// TwinCAT 3 PLC project PLC_1
// ProgramVersion: 3.1.4024.0
// libraries:
//   Tc2_Standard, * (Beckhoff Automation GmbH)
//   Tc2_System, * (Beckhoff Automation GmbH)
//   Tc2_XmlDataSrv, * (Beckhoff Automation GmbH)
//   Tc3_JsonXml, * (Beckhoff Automation GmbH)
//   Tc3_Module, * (Beckhoff Automation GmbH)
// project tree:
//   DUTs/GenericHierarchyList/GenericHierarchy/ItemCS/Content/DefaultIdentity/ St_DefaultIdentity.TcDUT
//   DUTs/GenericHierarchyList/GenericHierarchy/ItemCS/Content/ItemList/ItemOUT1/Content/DefaultIdentity/ ST_DefaultIdentityOUT1.TcDUT
//   DUTs/GenericHierarchyList/GenericHierarchy/ItemCS/Content/ItemList/ItemOUT1/Content/ItemList/ItemPK1/Identity/ ST_Identity_PK1_OUT1.TcDUT
//   DUTs/GenericHierarchyList/GenericHierarchy/ItemCS/Content/ItemList/ItemOUT1/Content/ItemList/ItemPK1/logs/ ST_logs_PK1_OUT1.TcDUT (not stored)
//   DUTs/GenericHierarchyList/GenericHierarchy/ItemCS/Content/ItemList/ItemOUT1/Content/ItemList/ItemPK1/RejectReason/ ST_RejectReason_PK1_OUT1.TcDUT
//   DUTs/GenericHierarchyList/GenericHierarchy/ItemCS/Content/ItemList/ItemOUT1/Content/ItemList/ItemPK1/ ST_ItemPK1_OUT1.TcDUT
//   DUTs/GenericHierarchyList/GenericHierarchy/ItemCS/Content/ItemList/ItemOUT1/Content/ItemList/ItemPK2/Identity/ ST_Identity_PK2_OUT1.TcDUT
//   DUTs/GenericHierarchyList/GenericHierarchy/ItemCS/Content/ItemList/ItemOUT1/Content/ItemList/ItemPK2/logs/ ST_logs_PK2_OUT1.TcDUT (not stored)
//   DUTs/GenericHierarchyList/GenericHierarchy/ItemCS/Content/ItemList/ItemOUT1/Content/ItemList/ItemPK2/RejectReason/ ST_RejectReason_PK2_OUT1.TcDUT
//   DUTs/GenericHierarchyList/GenericHierarchy/ItemCS/Content/ItemList/ItemOUT1/Content/ItemList/ItemPK2/ ST_ItemPK2_OUT1.TcDUT
//   DUTs/GenericHierarchyList/GenericHierarchy/ItemCS/Content/ItemList/ItemOUT1/Content/ItemList/ItemPK3/Identity/ ST_Identity_PK3_OUT1.TcDUT
//   DUTs/GenericHierarchyList/GenericHierarchy/ItemCS/Content/ItemList/ItemOUT1/Content/ItemList/ItemPK3/logs/ ST_logs_PK3_OUT1.TcDUT (not stored)
//   DUTs/GenericHierarchyList/GenericHierarchy/ItemCS/Content/ItemList/ItemOUT1/Content/ItemList/ItemPK3/RejectReason/ ST_RejectReason_PK3_OUT1.TcDUT
//   DUTs/GenericHierarchyList/GenericHierarchy/ItemCS/Content/ItemList/ItemOUT1/Content/ItemList/ItemPK3/ ST_ItemPK3_OUT1.TcDUT
//   DUTs/GenericHierarchyList/GenericHierarchy/ItemCS/Content/ItemList/ItemOUT1/Content/ItemList/ItemPK4/Identity/ ST_Identity_PK4_OUT1.TcDUT
//   DUTs/GenericHierarchyList/GenericHierarchy/ItemCS/Content/ItemList/ItemOUT1/Content/ItemList/ItemPK4/logs/ ST_logs_PK4_OUT1.TcDUT (not stored)
//   DUTs/GenericHierarchyList/GenericHierarchy/ItemCS/Content/ItemList/ItemOUT1/Content/ItemList/ItemPK4/RejectReason/ ST_RejectReason_PK4_OUT1.TcDUT
//   DUTs/GenericHierarchyList/GenericHierarchy/ItemCS/Content/ItemList/ItemOUT1/Content/ItemList/ItemPK4/ ST_ItemPK4_OUT1.TcDUT
//   DUTs/GenericHierarchyList/GenericHierarchy/ItemCS/Content/ItemList/ItemOUT1/Content/ItemList/ ST_ItemListOUT1.TcDUT
//   DUTs/GenericHierarchyList/GenericHierarchy/ItemCS/Content/ItemList/ItemOUT1/Content/ ST_ContentOUT1.TcDUT
//   DUTs/GenericHierarchyList/GenericHierarchy/ItemCS/Content/ItemList/ItemOUT1/Identity/ ST_IdentityOUT1.TcDUT
//   DUTs/GenericHierarchyList/GenericHierarchy/ItemCS/Content/ItemList/ItemOUT1/logs/ ST_logsOUT1.TcDUT (not stored)
//   DUTs/GenericHierarchyList/GenericHierarchy/ItemCS/Content/ItemList/ItemOUT1/RejectReason/ ST_RejectReasonOUT1.TcDUT
//   DUTs/GenericHierarchyList/GenericHierarchy/ItemCS/Content/ItemList/ItemOUT1/ ST_ItemOUT1.TcDUT
//   DUTs/GenericHierarchyList/GenericHierarchy/ItemCS/Content/ItemList/ItemOUT2/Content/DefaultIdentity/ ST_DefaultIdentityOUT2.TcDUT
//   DUTs/GenericHierarchyList/GenericHierarchy/ItemCS/Content/ItemList/ItemOUT2/Content/ItemList/ItemPK1/Identity/ ST_Identity_PK1_OUT2.TcDUT
//   DUTs/GenericHierarchyList/GenericHierarchy/ItemCS/Content/ItemList/ItemOUT2/Content/ItemList/ItemPK1/logs/ ST_logs_PK1_OUT2.TcDUT (not stored)
//   DUTs/GenericHierarchyList/GenericHierarchy/ItemCS/Content/ItemList/ItemOUT2/Content/ItemList/ItemPK1/RejectReason/ ST_RejectReason_PK1_OUT2.TcDUT
//   DUTs/GenericHierarchyList/GenericHierarchy/ItemCS/Content/ItemList/ItemOUT2/Content/ItemList/ItemPK1/ ST_ItemPK1_OUT2.TcDUT
//   DUTs/GenericHierarchyList/GenericHierarchy/ItemCS/Content/ItemList/ItemOUT2/Content/ItemList/ItemPK2/Identity/ ST_Identity_PK2_OUT2.TcDUT
//   DUTs/GenericHierarchyList/GenericHierarchy/ItemCS/Content/ItemList/ItemOUT2/Content/ItemList/ItemPK2/logs/ ST_logs_PK2_OUT2.TcDUT (not stored)
//   DUTs/GenericHierarchyList/GenericHierarchy/ItemCS/Content/ItemList/ItemOUT2/Content/ItemList/ItemPK2/RejectReason/ ST_RejectReason_PK2_OUT2.TcDUT
//   DUTs/GenericHierarchyList/GenericHierarchy/ItemCS/Content/ItemList/ItemOUT2/Content/ItemList/ItemPK2/ ST_ItemPK2_OUT2.TcDUT
//   DUTs/GenericHierarchyList/GenericHierarchy/ItemCS/Content/ItemList/ItemOUT2/Content/ItemList/ItemPK3/Identity/ ST_Identity_PK3_OUT2.TcDUT
//   DUTs/GenericHierarchyList/GenericHierarchy/ItemCS/Content/ItemList/ItemOUT2/Content/ItemList/ItemPK3/logs/ ST_logs_PK3_OUT2.TcDUT (not stored)
//   DUTs/GenericHierarchyList/GenericHierarchy/ItemCS/Content/ItemList/ItemOUT2/Content/ItemList/ItemPK3/RejectReason/ ST_RejectReason_PK3_OUT2.TcDUT
//   DUTs/GenericHierarchyList/GenericHierarchy/ItemCS/Content/ItemList/ItemOUT2/Content/ItemList/ItemPK3/ ST_ItemPK3_OUT2.TcDUT
//   DUTs/GenericHierarchyList/GenericHierarchy/ItemCS/Content/ItemList/ItemOUT2/Content/ItemList/ItemPK4/Identity/ ST_Identity_PK4_OUT2.TcDUT
//   DUTs/GenericHierarchyList/GenericHierarchy/ItemCS/Content/ItemList/ItemOUT2/Content/ItemList/ItemPK4/logs/ ST_logs_PK4_OUT2.TcDUT (not stored)
//   DUTs/GenericHierarchyList/GenericHierarchy/ItemCS/Content/ItemList/ItemOUT2/Content/ItemList/ItemPK4/RejectReason/ ST_RejectReason_PK4_OUT2.TcDUT
//   DUTs/GenericHierarchyList/GenericHierarchy/ItemCS/Content/ItemList/ItemOUT2/Content/ItemList/ItemPK4/ ST_ItemPK4_OUT2.TcDUT
//   DUTs/GenericHierarchyList/GenericHierarchy/ItemCS/Content/ItemList/ItemOUT2/Content/ItemList/ ST_ItemListOUT2.TcDUT
//   DUTs/GenericHierarchyList/GenericHierarchy/ItemCS/Content/ItemList/ItemOUT2/Content/ ST_ContentOUT2.TcDUT
//   DUTs/GenericHierarchyList/GenericHierarchy/ItemCS/Content/ItemList/ItemOUT2/Identity/ ST_IdentityOUT2.TcDUT
//   DUTs/GenericHierarchyList/GenericHierarchy/ItemCS/Content/ItemList/ItemOUT2/logs/ ST_logsOUT2.TcDUT (not stored)
//   DUTs/GenericHierarchyList/GenericHierarchy/ItemCS/Content/ItemList/ItemOUT2/RejectReason/ ST_RejectReasonOUT2.TcDUT
//   DUTs/GenericHierarchyList/GenericHierarchy/ItemCS/Content/ItemList/ItemOUT2/ ST_ItemOUT2.TcDUT
//   DUTs/GenericHierarchyList/GenericHierarchy/ItemCS/Content/ItemList/ItemOUT3/Content/DefaultIdentity/ ST_DefaultIdentityOUT3.TcDUT
//   DUTs/GenericHierarchyList/GenericHierarchy/ItemCS/Content/ItemList/ItemOUT3/Content/ItemList/ItemPK1/Identity/ ST_Identity_PK1_OUT3.TcDUT
//   DUTs/GenericHierarchyList/GenericHierarchy/ItemCS/Content/ItemList/ItemOUT3/Content/ItemList/ItemPK1/logs/ ST_logs_PK1_OUT3.TcDUT (not stored)
//   DUTs/GenericHierarchyList/GenericHierarchy/ItemCS/Content/ItemList/ItemOUT3/Content/ItemList/ItemPK1/RejectReason/ ST_RejectReason_PK1_OUT3.TcDUT
//   DUTs/GenericHierarchyList/GenericHierarchy/ItemCS/Content/ItemList/ItemOUT3/Content/ItemList/ItemPK1/ ST_ItemPK1_OUT3.TcDUT
//   DUTs/GenericHierarchyList/GenericHierarchy/ItemCS/Content/ItemList/ItemOUT3/Content/ItemList/ItemPK2/Identity/ ST_Identity_PK2_OUT3.TcDUT
//   DUTs/GenericHierarchyList/GenericHierarchy/ItemCS/Content/ItemList/ItemOUT3/Content/ItemList/ItemPK2/logs/ ST_logs_PK2_OUT3.TcDUT (not stored)
//   DUTs/GenericHierarchyList/GenericHierarchy/ItemCS/Content/ItemList/ItemOUT3/Content/ItemList/ItemPK2/RejectReason/ ST_RejectReason_PK2_OUT3.TcDUT
//   DUTs/GenericHierarchyList/GenericHierarchy/ItemCS/Content/ItemList/ItemOUT3/Content/ItemList/ItemPK2/ ST_ItemPK2_OUT3.TcDUT
//   DUTs/GenericHierarchyList/GenericHierarchy/ItemCS/Content/ItemList/ItemOUT3/Content/ItemList/ItemPK3/Identity/ ST_Identity_PK3_OUT3.TcDUT
//   DUTs/GenericHierarchyList/GenericHierarchy/ItemCS/Content/ItemList/ItemOUT3/Content/ItemList/ItemPK3/logs/ ST_logs_PK3_OUT3.TcDUT (not stored)
//   DUTs/GenericHierarchyList/GenericHierarchy/ItemCS/Content/ItemList/ItemOUT3/Content/ItemList/ItemPK3/RejectReason/ ST_RejectReason_PK3_OUT3.TcDUT
//   DUTs/GenericHierarchyList/GenericHierarchy/ItemCS/Content/ItemList/ItemOUT3/Content/ItemList/ItemPK3/ ST_ItemPK3_OUT3.TcDUT
//   DUTs/GenericHierarchyList/GenericHierarchy/ItemCS/Content/ItemList/ItemOUT3/Content/ItemList/ItemPK4/Identity/ ST_Identity_PK4_OUT3.TcDUT
//   DUTs/GenericHierarchyList/GenericHierarchy/ItemCS/Content/ItemList/ItemOUT3/Content/ItemList/ItemPK4/logs/ ST_logs_PK4_OUT3.TcDUT (not stored)
//   DUTs/GenericHierarchyList/GenericHierarchy/ItemCS/Content/ItemList/ItemOUT3/Content/ItemList/ItemPK4/RejectReason/ ST_RejectReason_PK4_OUT3.TcDUT
//   DUTs/GenericHierarchyList/GenericHierarchy/ItemCS/Content/ItemList/ItemOUT3/Content/ItemList/ItemPK4/ ST_ItemPK4_OUT3.TcDUT
//   DUTs/GenericHierarchyList/GenericHierarchy/ItemCS/Content/ItemList/ItemOUT3/Content/ItemList/ ST_ItemListOUT3.TcDUT
//   DUTs/GenericHierarchyList/GenericHierarchy/ItemCS/Content/ItemList/ItemOUT3/Content/ ST_ContentOUT3.TcDUT
//   DUTs/GenericHierarchyList/GenericHierarchy/ItemCS/Content/ItemList/ItemOUT3/Identity/ ST_IdentityOUT3.TcDUT
//   DUTs/GenericHierarchyList/GenericHierarchy/ItemCS/Content/ItemList/ItemOUT3/logs/ ST_logsOUT3.TcDUT (not stored)
//   DUTs/GenericHierarchyList/GenericHierarchy/ItemCS/Content/ItemList/ItemOUT3/RejectReason/ ST_RejectReasonOUT3.TcDUT
//   DUTs/GenericHierarchyList/GenericHierarchy/ItemCS/Content/ItemList/ItemOUT3/ ST_ItemOUT3.TcDUT
//   DUTs/GenericHierarchyList/GenericHierarchy/ItemCS/Content/ItemList/ ST_ItemList.TcDUT
//   DUTs/GenericHierarchyList/GenericHierarchy/ItemCS/Content/ ST_Content.TcDUT
//   DUTs/GenericHierarchyList/GenericHierarchy/ItemCS/Identity/ ST_Identity.TcDUT
//   DUTs/GenericHierarchyList/GenericHierarchy/ItemCS/logs/ ST_logs.TcDUT (not stored)
//   DUTs/GenericHierarchyList/GenericHierarchy/ItemCS/RejectReason/ ST_RejectReason.TcDUT
//   DUTs/GenericHierarchyList/GenericHierarchy/ItemCS/ ST_ItemCS.TcDUT
//   DUTs/GenericHierarchyList/GenericHierarchy/ ST_GenericHierarchy_Write.TcDUT
//   DUTs/GenericHierarchyList/Messageheader/ ST_MessageHeader_Write.TcDUT
//   DUTs/GenericHierarchyList/ ST_GenericHierarchyList.TcDUT
//   DUTs/ProductionChange/PRODUCTINFORMATION/PRODUCT/HIERARCHYDATALIST/HIERARCHYDATACS/ ST_HIERARCHYDATACS.TcDUT
//   DUTs/ProductionChange/PRODUCTINFORMATION/PRODUCT/HIERARCHYDATALIST/HIERARCHYDATAOUT/ ST_HIERARCHYDATAOUT.TcDUT
//   DUTs/ProductionChange/PRODUCTINFORMATION/PRODUCT/HIERARCHYDATALIST/HIERARCHYDATAPK/ ST_HIERARCHYDATAPK.TcDUT
//   DUTs/ProductionChange/PRODUCTINFORMATION/PRODUCT/HIERARCHYDATALIST/ ST_HIERARCHYDATALIST.TcDUT
//   DUTs/ProductionChange/PRODUCTINFORMATION/PRODUCT/ ST_PRODUCT.TcDUT
//   DUTs/ProductionChange/PRODUCTINFORMATION/SETTINGS/TOLERANCETHRESHOLDOUT/ ST_TOLERANCETHRESHOLDOUT.TcDUT
//   DUTs/ProductionChange/PRODUCTINFORMATION/SETTINGS/ ST_SETTINGS.TcDUT
//   DUTs/ProductionChange/PRODUCTINFORMATION/SETTINGS/TOLERANCETHRESHOLDPK/ ST_TOLERANCETHRESHOLDPK.TcDUT
//   DUTs/ProductionChange/PRODUCTINFORMATION/ ST_PRODUCTINFORMATION.TcDUT
//   DUTs/ProductionChange/ ST_MESSAGEHEADER.TcDUT, ST_ProductionChange.TcDUT
//   / PlcTask.TcTTO
//   POUs/ FB_XMLRead.TcPOU, FB_XmlWrite.TcPOU, MAIN.TcPOU
// real-time tasks:
//   TASK PlcTask: cycle T#10ms, priority 20, ADS port 350

CONFIGURATION PLC_1
    RESOURCE PLC ON TwinCAT3
        TASK PlcTask(INTERVAL := T#10ms, PRIORITY := 20);
        PROGRAM MAIN WITH PlcTask : MAIN;
    END_RESOURCE
END_CONFIGURATION

// ---- DUTs/GenericHierarchyList/GenericHierarchy/ItemCS/Content/DefaultIdentity/St_DefaultIdentity.TcDUT
TYPE St_DefaultIdentity :
STRUCT
	SKU					:STRING;
	GTIN				:STRING;
	ProductionOrder		:STRING;
	LocalProductionOrder:STRING;
	PITCode				:STRING;
	BatchID				:STRING;
	ProductionLine		:STRING;
END_STRUCT
END_TYPE

// ---- DUTs/GenericHierarchyList/GenericHierarchy/ItemCS/Content/ItemList/ItemOUT1/Content/DefaultIdentity/ST_DefaultIdentityOUT1.TcDUT
TYPE ST_DefaultIdentityOUT1 :
STRUCT
	SKU						:STRING;
	GTIN					:STRING;
	ProductionOrder			:STRING;
	LocalProductionOrder	:STRING;
	PITCode					:STRING;
	BatchID					:STRING;
	ProductionLine			:STRING;
END_STRUCT
END_TYPE

// ---- DUTs/GenericHierarchyList/GenericHierarchy/ItemCS/Content/ItemList/ItemOUT1/Content/ItemList/ItemPK1/Identity/ST_Identity_PK1_OUT1.TcDUT
TYPE ST_Identity_PK1_OUT1 :
STRUCT
	ID	:STRING;
	ReadQuality:STRING;
END_STRUCT
END_TYPE

// ---- DUTs/GenericHierarchyList/GenericHierarchy/ItemCS/Content/ItemList/ItemOUT1/Content/ItemList/ItemPK1/RejectReason/ST_RejectReason_PK1_OUT1.TcDUT
TYPE ST_RejectReason_PK1_OUT1 :
STRUCT
	Reason	:STRING;
END_STRUCT
END_TYPE

// ---- DUTs/GenericHierarchyList/GenericHierarchy/ItemCS/Content/ItemList/ItemOUT1/Content/ItemList/ItemPK1/ST_ItemPK1_OUT1.TcDUT
TYPE ST_ItemPK1_OUT1 :
STRUCT
	Identity		:ST_Identity_PK1_OUT1;
	ItemState		:STRING;
	RejectReason	:ST_RejectReason_PK1_OUT1;
	logs			:ST_logs_PK1_OUT1;
	NoRead			:STRING;
END_STRUCT
END_TYPE

// ---- DUTs/GenericHierarchyList/GenericHierarchy/ItemCS/Content/ItemList/ItemOUT1/Content/ItemList/ItemPK2/Identity/ST_Identity_PK2_OUT1.TcDUT
TYPE ST_Identity_PK2_OUT1 :
STRUCT
	ID	:STRING;
	ReadQuality:STRING;
END_STRUCT
END_TYPE

// ---- DUTs/GenericHierarchyList/GenericHierarchy/ItemCS/Content/ItemList/ItemOUT1/Content/ItemList/ItemPK2/RejectReason/ST_RejectReason_PK2_OUT1.TcDUT
TYPE ST_RejectReason_PK2_OUT1 :
STRUCT
	Reason	:STRING;
END_STRUCT
END_TYPE

// ---- DUTs/GenericHierarchyList/GenericHierarchy/ItemCS/Content/ItemList/ItemOUT1/Content/ItemList/ItemPK2/ST_ItemPK2_OUT1.TcDUT
TYPE ST_ItemPK2_OUT1 :
STRUCT
	Identity		:ST_Identity_PK2_OUT1;
	ItemState		:STRING;
	RejectReason	:ST_RejectReason_PK2_OUT1;
	logs			:ST_logs_PK2_OUT1;
	NoRead			:STRING;
END_STRUCT
END_TYPE

// ---- DUTs/GenericHierarchyList/GenericHierarchy/ItemCS/Content/ItemList/ItemOUT1/Content/ItemList/ItemPK3/Identity/ST_Identity_PK3_OUT1.TcDUT
TYPE ST_Identity_PK3_OUT1 :
STRUCT
	ID	:STRING;
	ReadQuality:STRING;
END_STRUCT
END_TYPE

// ---- DUTs/GenericHierarchyList/GenericHierarchy/ItemCS/Content/ItemList/ItemOUT1/Content/ItemList/ItemPK3/RejectReason/ST_RejectReason_PK3_OUT1.TcDUT
TYPE ST_RejectReason_PK3_OUT1 :
STRUCT
	Reason	:STRING;
END_STRUCT
END_TYPE

// ---- DUTs/GenericHierarchyList/GenericHierarchy/ItemCS/Content/ItemList/ItemOUT1/Content/ItemList/ItemPK3/ST_ItemPK3_OUT1.TcDUT
TYPE ST_ItemPK3_OUT1 :
STRUCT
	Identity		:ST_Identity_PK3_OUT1;
	ItemState		:STRING;
	RejectReason	:ST_RejectReason_PK3_OUT1;
	logs			:ST_logs_PK3_OUT1;
	NoRead			:STRING;
END_STRUCT
END_TYPE

// ---- DUTs/GenericHierarchyList/GenericHierarchy/ItemCS/Content/ItemList/ItemOUT1/Content/ItemList/ItemPK4/Identity/ST_Identity_PK4_OUT1.TcDUT
TYPE ST_Identity_PK4_OUT1 :
STRUCT
	ID	:STRING;
	ReadQuality:STRING;
END_STRUCT
END_TYPE

// ---- DUTs/GenericHierarchyList/GenericHierarchy/ItemCS/Content/ItemList/ItemOUT1/Content/ItemList/ItemPK4/RejectReason/ST_RejectReason_PK4_OUT1.TcDUT
TYPE ST_RejectReason_PK4_OUT1 :
STRUCT
	Reason	:STRING;
END_STRUCT
END_TYPE

// ---- DUTs/GenericHierarchyList/GenericHierarchy/ItemCS/Content/ItemList/ItemOUT1/Content/ItemList/ItemPK4/ST_ItemPK4_OUT1.TcDUT
TYPE ST_ItemPK4_OUT1 :
STRUCT
	Identity		:ST_Identity_PK4_OUT1;
	ItemState		:STRING;
	RejectReason	:ST_RejectReason_PK4_OUT1;
	logs			:ST_logs_PK4_OUT1;
	NoRead			:STRING;
END_STRUCT
END_TYPE

// ---- DUTs/GenericHierarchyList/GenericHierarchy/ItemCS/Content/ItemList/ItemOUT1/Content/ItemList/ST_ItemListOUT1.TcDUT
TYPE ST_ItemListOUT1 :
STRUCT
	ItemPK1 	:ST_ItemPK1_OUT1;
	ItemPK2 	:ST_ItemPK2_OUT1;
	ItemPK3 	:ST_ItemPK3_OUT1;
	ItemPK4 	:ST_ItemPK4_OUT1;
END_STRUCT
END_TYPE

// ---- DUTs/GenericHierarchyList/GenericHierarchy/ItemCS/Content/ItemList/ItemOUT1/Content/ST_ContentOUT1.TcDUT
TYPE ST_ContentOUT1 :
STRUCT
	DefaultIdentity   :ST_DefaultIdentityOUT1;
	ExpectedItemCount	:STRING;
	ItemReadRate		:STRING;
	ItemList			:ST_ItemListOUT1;
END_STRUCT
END_TYPE

// ---- DUTs/GenericHierarchyList/GenericHierarchy/ItemCS/Content/ItemList/ItemOUT1/Identity/ST_IdentityOUT1.TcDUT
TYPE ST_IdentityOUT1 :
STRUCT
	ID	:STRING;
	ReadQuality:STRING;
END_STRUCT
END_TYPE

// ---- DUTs/GenericHierarchyList/GenericHierarchy/ItemCS/Content/ItemList/ItemOUT1/RejectReason/ST_RejectReasonOUT1.TcDUT
TYPE ST_RejectReasonOUT1 :
STRUCT
	Reason	:STRING;
END_STRUCT
END_TYPE

// ---- DUTs/GenericHierarchyList/GenericHierarchy/ItemCS/Content/ItemList/ItemOUT1/ST_ItemOUT1.TcDUT
TYPE ST_ItemOUT1 :
STRUCT
	Identity		:ST_IdentityOUT1;
	ItemState		:STRING;
	RejectReason	:ST_RejectReasonOUT1;
	logs			:ST_logsOUT1;
	NoRead			:STRING;
	Content			:ST_ContentOUT1;
END_STRUCT
END_TYPE

// ---- DUTs/GenericHierarchyList/GenericHierarchy/ItemCS/Content/ItemList/ItemOUT2/Content/DefaultIdentity/ST_DefaultIdentityOUT2.TcDUT
TYPE ST_DefaultIdentityOUT2 :
STRUCT
	SKU						:STRING;
	GTIN					:STRING;
	ProductionOrder			:STRING;
	LocalProductionOrder	:STRING;
	PITCode					:STRING;
	BatchID					:STRING;
	ProductionLine			:STRING;
END_STRUCT
END_TYPE

// ---- DUTs/GenericHierarchyList/GenericHierarchy/ItemCS/Content/ItemList/ItemOUT2/Content/ItemList/ItemPK1/Identity/ST_Identity_PK1_OUT2.TcDUT
TYPE ST_Identity_PK1_OUT2 :
STRUCT
	ID	:STRING;
	ReadQuality:STRING;
END_STRUCT
END_TYPE

// ---- DUTs/GenericHierarchyList/GenericHierarchy/ItemCS/Content/ItemList/ItemOUT2/Content/ItemList/ItemPK1/RejectReason/ST_RejectReason_PK1_OUT2.TcDUT
TYPE ST_RejectReason_PK1_OUT2 :
STRUCT
	Reason	:STRING;
END_STRUCT
END_TYPE

// ---- DUTs/GenericHierarchyList/GenericHierarchy/ItemCS/Content/ItemList/ItemOUT2/Content/ItemList/ItemPK1/ST_ItemPK1_OUT2.TcDUT
TYPE ST_ItemPK1_OUT2 :
STRUCT
	Identity		:ST_Identity_PK1_OUT2;
	ItemState		:STRING;
	RejectReason	:ST_RejectReason_PK1_OUT2;
	logs			:ST_logs_PK1_OUT2;
	NoRead			:STRING;
END_STRUCT
END_TYPE

// ---- DUTs/GenericHierarchyList/GenericHierarchy/ItemCS/Content/ItemList/ItemOUT2/Content/ItemList/ItemPK2/Identity/ST_Identity_PK2_OUT2.TcDUT
TYPE ST_Identity_PK2_OUT2 :
STRUCT
	ID	:STRING;
	ReadQuality:STRING;
END_STRUCT
END_TYPE

// ---- DUTs/GenericHierarchyList/GenericHierarchy/ItemCS/Content/ItemList/ItemOUT2/Content/ItemList/ItemPK2/RejectReason/ST_RejectReason_PK2_OUT2.TcDUT
TYPE ST_RejectReason_PK2_OUT2 :
STRUCT
	Reason	:STRING;
END_STRUCT
END_TYPE

// ---- DUTs/GenericHierarchyList/GenericHierarchy/ItemCS/Content/ItemList/ItemOUT2/Content/ItemList/ItemPK2/ST_ItemPK2_OUT2.TcDUT
TYPE ST_ItemPK2_OUT2 :
STRUCT
	Identity		:ST_Identity_PK2_OUT2;
	ItemState		:STRING;
	RejectReason	:ST_RejectReason_PK2_OUT2;
	logs			:ST_logs_PK2_OUT2;
	NoRead			:STRING;
END_STRUCT
END_TYPE

// ---- DUTs/GenericHierarchyList/GenericHierarchy/ItemCS/Content/ItemList/ItemOUT2/Content/ItemList/ItemPK3/Identity/ST_Identity_PK3_OUT2.TcDUT
TYPE ST_Identity_PK3_OUT2 :
STRUCT
	ID	:STRING;
	ReadQuality:STRING;
END_STRUCT
END_TYPE

// ---- DUTs/GenericHierarchyList/GenericHierarchy/ItemCS/Content/ItemList/ItemOUT2/Content/ItemList/ItemPK3/RejectReason/ST_RejectReason_PK3_OUT2.TcDUT
TYPE ST_RejectReason_PK3_OUT2 :
STRUCT
	Reason	:STRING;
END_STRUCT
END_TYPE

// ---- DUTs/GenericHierarchyList/GenericHierarchy/ItemCS/Content/ItemList/ItemOUT2/Content/ItemList/ItemPK3/ST_ItemPK3_OUT2.TcDUT
TYPE ST_ItemPK3_OUT2 :
STRUCT
	Identity		:ST_Identity_PK3_OUT2;
	ItemState		:STRING;
	RejectReason	:ST_RejectReason_PK3_OUT2;
	logs			:ST_logs_PK3_OUT2;
	NoRead			:STRING;
END_STRUCT
END_TYPE

// ---- DUTs/GenericHierarchyList/GenericHierarchy/ItemCS/Content/ItemList/ItemOUT2/Content/ItemList/ItemPK4/Identity/ST_Identity_PK4_OUT2.TcDUT
TYPE ST_Identity_PK4_OUT2 :
STRUCT
	ID	:STRING;
	ReadQuality:STRING;
END_STRUCT
END_TYPE

// ---- DUTs/GenericHierarchyList/GenericHierarchy/ItemCS/Content/ItemList/ItemOUT2/Content/ItemList/ItemPK4/RejectReason/ST_RejectReason_PK4_OUT2.TcDUT
TYPE ST_RejectReason_PK4_OUT2 :
STRUCT
	Reason	:STRING;
END_STRUCT
END_TYPE

// ---- DUTs/GenericHierarchyList/GenericHierarchy/ItemCS/Content/ItemList/ItemOUT2/Content/ItemList/ItemPK4/ST_ItemPK4_OUT2.TcDUT
TYPE ST_ItemPK4_OUT2 :
STRUCT
	Identity		:ST_Identity_PK4_OUT2;
	ItemState		:STRING;
	RejectReason	:ST_RejectReason_PK4_OUT2;
	logs			:ST_logs_PK4_OUT2;
	NoRead			:STRING;
END_STRUCT
END_TYPE

// ---- DUTs/GenericHierarchyList/GenericHierarchy/ItemCS/Content/ItemList/ItemOUT2/Content/ItemList/ST_ItemListOUT2.TcDUT
TYPE ST_ItemListOUT2 :
STRUCT
	ItemPK1 	:ST_ItemPK1_OUT2;
	ItemPK2 	:ST_ItemPK2_OUT2;
	ItemPK3 	:ST_ItemPK3_OUT2;
	ItemPK4 	:ST_ItemPK4_OUT2;
END_STRUCT
END_TYPE

// ---- DUTs/GenericHierarchyList/GenericHierarchy/ItemCS/Content/ItemList/ItemOUT2/Content/ST_ContentOUT2.TcDUT
TYPE ST_ContentOUT2 :
STRUCT
	DefaultIdentity   :ST_DefaultIdentityOUT2;
	ExpectedItemCount	:STRING;
	ItemReadRate		:STRING;
	ItemList			:ST_ItemListOUT2;
END_STRUCT
END_TYPE

// ---- DUTs/GenericHierarchyList/GenericHierarchy/ItemCS/Content/ItemList/ItemOUT2/Identity/ST_IdentityOUT2.TcDUT
TYPE ST_IdentityOUT2 :
STRUCT
	ID	:STRING;
	ReadQuality:STRING;
END_STRUCT
END_TYPE

// ---- DUTs/GenericHierarchyList/GenericHierarchy/ItemCS/Content/ItemList/ItemOUT2/RejectReason/ST_RejectReasonOUT2.TcDUT
TYPE ST_RejectReasonOUT2 :
STRUCT
	Reason	:STRING;
END_STRUCT
END_TYPE

// ---- DUTs/GenericHierarchyList/GenericHierarchy/ItemCS/Content/ItemList/ItemOUT2/ST_ItemOUT2.TcDUT
TYPE ST_ItemOUT2 :
STRUCT
	Identity		:ST_IdentityOUT2;
	ItemState		:STRING;
	RejectReason	:ST_RejectReasonOUT2;
	logs			:ST_logsOUT2;
	NoRead			:STRING;
	Content			:ST_ContentOUT2;
END_STRUCT
END_TYPE

// ---- DUTs/GenericHierarchyList/GenericHierarchy/ItemCS/Content/ItemList/ItemOUT3/Content/DefaultIdentity/ST_DefaultIdentityOUT3.TcDUT
TYPE ST_DefaultIdentityOUT3 :
STRUCT
	SKU						:STRING;
	GTIN					:STRING;
	ProductionOrder			:STRING;
	LocalProductionOrder	:STRING;
	PITCode					:STRING;
	BatchID					:STRING;
	ProductionLine			:STRING;
END_STRUCT
END_TYPE

// ---- DUTs/GenericHierarchyList/GenericHierarchy/ItemCS/Content/ItemList/ItemOUT3/Content/ItemList/ItemPK1/Identity/ST_Identity_PK1_OUT3.TcDUT
TYPE ST_Identity_PK1_OUT3 :
STRUCT
	ID	:STRING;
	ReadQuality:STRING;
END_STRUCT
END_TYPE

// ---- DUTs/GenericHierarchyList/GenericHierarchy/ItemCS/Content/ItemList/ItemOUT3/Content/ItemList/ItemPK1/RejectReason/ST_RejectReason_PK1_OUT3.TcDUT
TYPE ST_RejectReason_PK1_OUT3 :
STRUCT
	Reason	:STRING;
END_STRUCT
END_TYPE

// ---- DUTs/GenericHierarchyList/GenericHierarchy/ItemCS/Content/ItemList/ItemOUT3/Content/ItemList/ItemPK1/ST_ItemPK1_OUT3.TcDUT
TYPE ST_ItemPK1_OUT3 :
STRUCT
	Identity		:ST_Identity_PK1_OUT3;
	ItemState		:STRING;
	RejectReason	:ST_RejectReason_PK1_OUT3;
	logs			:ST_logs_PK1_OUT3;
	NoRead			:STRING;
END_STRUCT
END_TYPE

// ---- DUTs/GenericHierarchyList/GenericHierarchy/ItemCS/Content/ItemList/ItemOUT3/Content/ItemList/ItemPK2/Identity/ST_Identity_PK2_OUT3.TcDUT
TYPE ST_Identity_PK2_OUT3 :
STRUCT
	ID	:STRING;
	ReadQuality:STRING;
END_STRUCT
END_TYPE

// ---- DUTs/GenericHierarchyList/GenericHierarchy/ItemCS/Content/ItemList/ItemOUT3/Content/ItemList/ItemPK2/RejectReason/ST_RejectReason_PK2_OUT3.TcDUT
TYPE ST_RejectReason_PK2_OUT3:
STRUCT
	Reason	:STRING;
END_STRUCT
END_TYPE

// ---- DUTs/GenericHierarchyList/GenericHierarchy/ItemCS/Content/ItemList/ItemOUT3/Content/ItemList/ItemPK2/ST_ItemPK2_OUT3.TcDUT
TYPE ST_ItemPK2_OUT3 :
STRUCT
	Identity		:ST_Identity_PK2_OUT3;
	ItemState		:STRING;
	RejectReason	:ST_RejectReason_PK2_OUT3;
	logs			:ST_logs_PK2_OUT3;
	NoRead			:STRING;
END_STRUCT
END_TYPE

// ---- DUTs/GenericHierarchyList/GenericHierarchy/ItemCS/Content/ItemList/ItemOUT3/Content/ItemList/ItemPK3/Identity/ST_Identity_PK3_OUT3.TcDUT
TYPE ST_Identity_PK3_OUT3 :
STRUCT
	ID	:STRING;
	ReadQuality:STRING;
END_STRUCT
END_TYPE

// ---- DUTs/GenericHierarchyList/GenericHierarchy/ItemCS/Content/ItemList/ItemOUT3/Content/ItemList/ItemPK3/RejectReason/ST_RejectReason_PK3_OUT3.TcDUT
TYPE ST_RejectReason_PK3_OUT3 :
STRUCT
	Reason	:STRING;
END_STRUCT
END_TYPE

// ---- DUTs/GenericHierarchyList/GenericHierarchy/ItemCS/Content/ItemList/ItemOUT3/Content/ItemList/ItemPK3/ST_ItemPK3_OUT3.TcDUT
TYPE ST_ItemPK3_OUT3 :
STRUCT
	Identity		:ST_Identity_PK3_OUT3;
	ItemState		:STRING;
	RejectReason	:ST_RejectReason_PK3_OUT3;
	logs			:ST_logs_PK3_OUT3;
	NoRead			:STRING;
END_STRUCT
END_TYPE

// ---- DUTs/GenericHierarchyList/GenericHierarchy/ItemCS/Content/ItemList/ItemOUT3/Content/ItemList/ItemPK4/Identity/ST_Identity_PK4_OUT3.TcDUT
TYPE ST_Identity_PK4_OUT3 :
STRUCT
	ID	:STRING;
	ReadQuality:STRING;
END_STRUCT
END_TYPE

// ---- DUTs/GenericHierarchyList/GenericHierarchy/ItemCS/Content/ItemList/ItemOUT3/Content/ItemList/ItemPK4/RejectReason/ST_RejectReason_PK4_OUT3.TcDUT
TYPE ST_RejectReason_PK4_OUT3 :
STRUCT
	Reason	:STRING;
END_STRUCT
END_TYPE

// ---- DUTs/GenericHierarchyList/GenericHierarchy/ItemCS/Content/ItemList/ItemOUT3/Content/ItemList/ItemPK4/ST_ItemPK4_OUT3.TcDUT
TYPE ST_ItemPK4_OUT3 :
STRUCT
	Identity		:ST_Identity_PK4_OUT3;
	ItemState		:STRING;
	RejectReason	:ST_RejectReason_PK4_OUT3;
	logs			:ST_logs_PK4_OUT3;
	NoRead			:STRING;
END_STRUCT
END_TYPE

// ---- DUTs/GenericHierarchyList/GenericHierarchy/ItemCS/Content/ItemList/ItemOUT3/Content/ItemList/ST_ItemListOUT3.TcDUT
TYPE ST_ItemListOUT3 :
STRUCT
	ItemPK1 	:ST_ItemPK1_OUT3;
	ItemPK2 	:ST_ItemPK2_OUT3;
	ItemPK3 	:ST_ItemPK3_OUT3;
	ItemPK4 	:ST_ItemPK4_OUT3;
END_STRUCT
END_TYPE

// ---- DUTs/GenericHierarchyList/GenericHierarchy/ItemCS/Content/ItemList/ItemOUT3/Content/ST_ContentOUT3.TcDUT
TYPE ST_ContentOUT3 :
STRUCT
	DefaultIdentity   :ST_DefaultIdentityOUT3;
	ExpectedItemCount	:STRING;
	ItemReadRate		:STRING;
	ItemList			:ST_ItemListOUT3;
END_STRUCT
END_TYPE

// ---- DUTs/GenericHierarchyList/GenericHierarchy/ItemCS/Content/ItemList/ItemOUT3/Identity/ST_IdentityOUT3.TcDUT
TYPE ST_IdentityOUT3 :
STRUCT
	ID	:STRING;
	ReadQuality:STRING;
END_STRUCT
END_TYPE

// ---- DUTs/GenericHierarchyList/GenericHierarchy/ItemCS/Content/ItemList/ItemOUT3/RejectReason/ST_RejectReasonOUT3.TcDUT
TYPE ST_RejectReasonOUT3 :
STRUCT
	Reason	:STRING;
END_STRUCT
END_TYPE

// ---- DUTs/GenericHierarchyList/GenericHierarchy/ItemCS/Content/ItemList/ItemOUT3/ST_ItemOUT3.TcDUT
TYPE ST_ItemOUT3 :
STRUCT
	Identity		:ST_IdentityOUT3;
	ItemState		:STRING;
	RejectReason	:ST_RejectReasonOUT3;
	logs			:ST_logsOUT3;
	NoRead			:STRING;
	Content			:ST_ContentOUT3;
END_STRUCT
END_TYPE

// ---- DUTs/GenericHierarchyList/GenericHierarchy/ItemCS/Content/ItemList/ST_ItemList.TcDUT
TYPE ST_ItemList :
STRUCT
	ItemOUT1	:ST_ItemOUT1;
	ItemOUT2	:ST_ItemOUT2;
	ItemOUT3	:ST_ItemOUT3;

END_STRUCT
END_TYPE

// ---- DUTs/GenericHierarchyList/GenericHierarchy/ItemCS/Content/ST_Content.TcDUT
TYPE ST_Content :
STRUCT
	DefaultIdentity		:St_DefaultIdentity;
	ExpectedItemCount	:STRING;
	ItemReadRate		:STRING;
	ItemList			:ST_ItemList;	
END_STRUCT
END_TYPE

// ---- DUTs/GenericHierarchyList/GenericHierarchy/ItemCS/Identity/ST_Identity.TcDUT
TYPE ST_Identity :
STRUCT
	SKU		:STRING;
	GTIN	:STRING;
	ID		:STRING;
	ReadQuality :STRING;
END_STRUCT
END_TYPE

// ---- DUTs/GenericHierarchyList/GenericHierarchy/ItemCS/RejectReason/ST_RejectReason.TcDUT
TYPE ST_RejectReason :
STRUCT
	Reason	:STRING;
END_STRUCT
END_TYPE

// ---- DUTs/GenericHierarchyList/GenericHierarchy/ItemCS/ST_ItemCS.TcDUT
TYPE ST_ItemCS :
STRUCT
	Identity		:ST_Identity;
	ItemState		:STRING;
	RejectReason	:ST_RejectReason;
	logs			:ST_logs;
	NoRead			:STRING;
	Content			:ST_Content;
	ProductionOrder		:STRING;
	LocalProductionOrder:STRING;
	PITCode				:STRING;
	BatchID				:STRING;
	ProductionLine		:STRING;
END_STRUCT
END_TYPE

// ---- DUTs/GenericHierarchyList/GenericHierarchy/ST_GenericHierarchy_Write.TcDUT
TYPE ST_GenericHierarchy_Write :
STRUCT
	HierarchyType		:STRING;
	_ACTION				:STRING;
	TrackingLevels		:STRING;
	TrackingIndicator	:STRING;
	ItemCS				:ST_ItemCS;
END_STRUCT
END_TYPE

// ---- DUTs/GenericHierarchyList/Messageheader/ST_MessageHeader_Write.TcDUT
TYPE ST_MessageHeader_Write :
STRUCT
	ReferenceID		:	STRING;
	CreationTimeLocalUTC	:	STRING;
	MessageType		:	STRING;
	SenderSystem	:	STRING;
	ReceiverSystem	:	STRING;
END_STRUCT
END_TYPE

// ---- DUTs/GenericHierarchyList/ST_GenericHierarchyList.TcDUT
TYPE ST_GenericHierarchyList :
STRUCT
	MessageHeader 		: 	ST_MessageHeader_Write;
	Factory 			: 	STRING;
	GenericHierarchy	:	ST_GenericHierarchy_Write;
	Attributes			:	STRING;
END_STRUCT
END_TYPE

// ---- DUTs/ProductionChange/PRODUCTINFORMATION/PRODUCT/HIERARCHYDATALIST/HIERARCHYDATACS/ST_HIERARCHYDATACS.TcDUT
TYPE ST_HIERARCHYDATACS :
STRUCT
	UNITQTY		:STRING;
	GTIN		:STRING;
	EAN			:STRING;
END_STRUCT
END_TYPE

// ---- DUTs/ProductionChange/PRODUCTINFORMATION/PRODUCT/HIERARCHYDATALIST/HIERARCHYDATAOUT/ST_HIERARCHYDATAOUT.TcDUT
TYPE ST_HIERARCHYDATAOUT :
STRUCT
	UNITQTY		:STRING;
	GTIN		:STRING;
	EAN			:STRING;
END_STRUCT
END_TYPE

// ---- DUTs/ProductionChange/PRODUCTINFORMATION/PRODUCT/HIERARCHYDATALIST/HIERARCHYDATAPK/ST_HIERARCHYDATAPK.TcDUT
TYPE ST_HIERARCHYDATAPK :
STRUCT
	UNITQTY		:STRING;
	GTIN		:STRING;
	EAN			:STRING;
END_STRUCT
END_TYPE

// ---- DUTs/ProductionChange/PRODUCTINFORMATION/PRODUCT/HIERARCHYDATALIST/ST_HIERARCHYDATALIST.TcDUT
TYPE ST_HIERARCHYDATALIST :
STRUCT
	TRACKINGLEVELS		:STRING;
	HIERARCHYDATAPK		:ST_HIERARCHYDATAPK;
	HIERARCHYDATAOUT	:ST_HIERARCHYDATAOUT;
	HIERARCHYDATACS		:ST_HIERARCHYDATACS;
END_STRUCT
END_TYPE

// ---- DUTs/ProductionChange/PRODUCTINFORMATION/PRODUCT/ST_PRODUCT.TcDUT
TYPE ST_PRODUCT :
STRUCT
	BATCHID				:STRING;
	PRODUCTIONORDER		:STRING;
	PITCODE				:STRING;
	HIERARCHYDATALIST	:ST_HIERARCHYDATALIST;
	UOM					:STRING;
END_STRUCT
END_TYPE

// ---- DUTs/ProductionChange/PRODUCTINFORMATION/SETTINGS/TOLERANCETHRESHOLDOUT/ST_TOLERANCETHRESHOLDOUT.TcDUT
TYPE ST_TOLERANCETHRESHOLDOUT :
STRUCT
	GOODREADPERCENTAGECS	:STRING;
END_STRUCT
END_TYPE

// ---- DUTs/ProductionChange/PRODUCTINFORMATION/SETTINGS/ST_SETTINGS.TcDUT
TYPE ST_SETTINGS :
STRUCT
	TOLERANCETHRESHOLDPK	:ST_TOLERANCETHRESHOLDPK;
	TOLERANCETHRESHOLDOUT	:ST_TOLERANCETHRESHOLDOUT;
END_STRUCT
END_TYPE

// ---- DUTs/ProductionChange/PRODUCTINFORMATION/SETTINGS/TOLERANCETHRESHOLDPK/ST_TOLERANCETHRESHOLDPK.TcDUT
TYPE ST_TOLERANCETHRESHOLDPK :
STRUCT
	GOODREADPERCENTAGECS	:STRING;
	GOODREADPERCENTAGEOUT	:STRING;
END_STRUCT
END_TYPE

// ---- DUTs/ProductionChange/PRODUCTINFORMATION/ST_PRODUCTINFORMATION.TcDUT
TYPE ST_PRODUCTINFORMATION :
STRUCT
	LINEID				:STRING;
	LINESYSTEMNO		:STRING;
	TRACKINGINDICATOR	:STRING;
	PRODUCTNO			:STRING;
	DESCRIPTION			:STRING;
	SETTINGS			:ST_SETTINGS;
	PRODUCT				:STRING;
END_STRUCT
END_TYPE

// ---- DUTs/ProductionChange/ST_MESSAGEHEADER.TcDUT
TYPE ST_MESSAGEHEADER :
STRUCT
	CREATIONDATE	:STRING;
	CREATIONTIME	:STRING;
	MESSAGETYPE		:STRING;
	TESTINDICATOR	:STRING;
	SENDERSYSTEM	:STRING;
	RECEIVERSYSTEM	:STRING;
	REFERENCEID		:STRING;
	SOURCEID		:STRING;
END_STRUCT
END_TYPE

// ---- DUTs/ProductionChange/ST_ProductionChange.TcDUT
TYPE ST_ProductionChange :
STRUCT
	MESSAGEHEADER  				: ST_MESSAGEHEADER;
	PRODUCTINFORMATION 			: ST_PRODUCTINFORMATION;
	PRODUCT						: ST_PRODUCT;
END_STRUCT
END_TYPE

// ---- POUs/MAIN.TcPOU
PROGRAM MAIN
VAR
	fbXmlRead	:	FB_XMLRead;
	fbXmlWrite	:	FB_XmlWrite;
END_VAR

fbXmlRead();
fbXmlWrite();

END_PROGRAM

// ---- POUs/FB_XMLRead.TcPOU
FUNCTION_BLOCK FB_XMLRead
VAR
	fbXmlSrvRead				:	FB_XmlSrvRead;
	fbXmlSrvReadByName			:	FB_XmlSrvReadByName;
	xExecute					:	BOOL:=FALSE;
	
	sFilePath					:T_MaxString := 'C:\Users\Ignacy\Downloads\PCM_Template.xml';
	sXPath						:T_MaxString := '/ProductionChange/MESSAGEHEADER';
	sXPath1						:T_MaxString := '/ProductionChange/PRODUCTINFORMATION';
	iStep						:INT;
	st_productionchange			:ST_ProductionChange;
END_VAR

fbXmlSrvRead(
   		sNetId := '', 
    	pSymAddr := ADR(st_productionchange.MESSAGEHEADER),
  		cbSymSize := SIZEOF(st_productionchange.MESSAGEHEADER),
    	sFilePath := sFilePath,
    	sXPath := sXPath,
    	bExecute := xExecute);
fbXmlSrvRead(
    	sNetId := '', 
    	pSymAddr := ADR(st_productionchange.PRODUCTINFORMATION),
   		cbSymSize := SIZEOF(st_productionchange.PRODUCTINFORMATION),
    	sFilePath := sFilePath,
    	sXPath := sXPath1,
    	bExecute := xExecute);

	IF NOT xExecute THEN
  	  xExecute := TRUE;
	END_IF;

	IF NOT fbXmlSrvRead.bBusy AND xExecute THEN
   	 xExecute := FALSE; 
	END_IF;

END_FUNCTION_BLOCK

// ---- POUs/FB_XmlWrite.TcPOU
FUNCTION_BLOCK FB_XmlWrite
VAR
	    // Obiekty XML
    fbXml                : FB_XmlDomParser;
    objRoot              : SXmlNode;
    objGenericHierachyList : SXmlNode;
	objAttributeXSD		:	SXmlNode;
  	objAttributeXSI		:	SXmlNode;
    // Atrybuty XML
    objAttribute         : SXmlAttribute;
    sXmlString           : STRING(1000); // Przechowywanie XML w postaci tekstowej

    // Flagi kontrolne
    xCreate              : BOOL := FALSE; // Flaga inicjalizacji tworzenia XML
    iFileWriteStep       : INT := 0;      // Kroki zapisu pliku
	xBusy : BOOL := FALSE;  
    // Operacje na plikach
    fbFileOpen           : FB_FileOpen;   // Otwieranie pliku
    fbFileClose          : FB_FileClose;  // Zamykanie pliku
    fbFileWrite          : FB_FileWrite;  // Zapis pliku
    uiFileHandle         : UINT := 0;     // Uchwyt pliku
    sFilePath            : STRING(255) := 'C:\Users\Ignacy\Desktop\CHM_Temp.xml'; // Ścieżka do pliku
	
	
	
	
	
	
	
	
	GenericHierarchyList	:	ST_GenericHierarchyList;
	fbxmlwrite	:	FB_XmlSrvWrite;
	xExecute	: 	BOOL;
	sXPathWrite		:T_MaxString:='/GenericHierarchyList';
END_VAR

IF xCreate THEN
  objRoot := fbXml.GetDocumentNode();
  // Root tree
  objGenericHierachyList := fbXml.AppendNode(objRoot, 'GenericHierarchyList');
  objAttributeXSD := fbXml.AppendAttribute(objGenericHierachyList, 'xmlns:xsd', 'http://www.w3.org/2001/XMLSchema');
  objAttributeXSI := fbXml.AppendAttribute(objGenericHierachyList, 'xmlns:xsi', 'http://www.w3.org/2001/XMLSchema-instance');
  fbXml.CopyDocument(sXmlString, SIZEOF(sXmlString)); // Zapisuje XML w zmiennej `sXmlString`
END_IF

uiFileHandle:=fbFileOpen.hFile;

CASE iFileWriteStep OF 
    0: // Waiting for execute
        IF xCreate THEN
			fbFileOpen.bExecute := TRUE;
            xCreate := FALSE; // Reset execute 
        END_IF
		
		IF fbFileOpen.bBusy THEN
            iFileWriteStep := 1; // Go to step 1
		END_IF

    1: // Reset xExecute and wait for xBusy reset
        fbFileOpen(bExecute := FALSE); // Stopping opening of file
        IF NOT fbFileOpen.bBusy THEN  
           iFileWriteStep := 2; // Go to step 2
        END_IF
	
    
    2: // Writing to file
// Lenght of string
		fbFileWrite.bExecute := TRUE;
		IF fbFileWrite.bBusy THEN
            iFileWriteStep := 3; // Go to step 3
		END_IF

    3:
        fbFileWrite(bExecute := FALSE); // Stop writing 
        IF NOT xBusy THEN
                iFileWriteStep := 4; // Go to step 0
        END_IF
	4:
		fbFileClose.bExecute := TRUE;
		IF fbFileClose.bBusy THEN
			iFileWriteStep := 5;
		END_IF
	5:
		fbFileClose.bExecute := FALSE;
		IF NOT fbFileClose.bBusy THEN
			iFileWriteStep := 0;
		END_IF
END_CASE

fbFileOpen(
                sNetId := '', 
                sPathName := sFilePath, 
                ePath := PATH_GENERIC, 
                nMode := FOPEN_MODEWRITE OR FOPEN_MODEPLUS, //modeplus
                bExecute := , 
                tTimeout := T#2S, 
                bBusy => xBusy, 
                bError =>, 
                nErrId =>, 
                hFile => uiFileHandle
            );
fbFileWrite(
	sNetId:='' , 
	hFile:=uiFileHandle , 
	pWriteBuff:=ADR(sXmlString)  , 
	cbWriteLen:=LEN(sXmlString) , 
	bExecute:= , 
	cbWrite=> );

fbFileClose(
	sNetId:= '', 
	hFile:=uiFileHandle , 
	bExecute:= , 
	tTimeout:=T#2S , 
	bBusy=> , 
	bError=> , 
	nErrId=> );
	
	
	
	
	
	
	
IF xExecute  THEN
   // Przygotowanie bExecute i ustawienie wartości
   fbxmlwrite.bExecute := TRUE;
   xExecute := FALSE; // Reset xExecute, aby uniknąć wielokrotnego wykonania
END_IF

// Wywołanie FB_XmlSrvWrite
fbxmlwrite(
    nMode := XMLSRV_ADDMISSING,        // Tryb dodawania brakujących elementów
    pSymAddr := ADR(GenericHierarchyList),         // Adres zmiennej struktury
    cbSymSize := SIZEOF(GenericHierarchyList),     // Rozmiar struktury
    sFilePath := sFilePath,       // Ścieżka do pliku XML
    sXPath := sXPathWrite,             // Ścieżka XPath do elementu
    bExecute := fbxmlwrite.bExecute    // Ustawienie flagi wykonania
);

// Reset bExecute po zakończeniu operacji
IF fbxmlwrite.bBusy THEN
   fbxmlwrite.bExecute := FALSE;
END_IF

END_FUNCTION_BLOCK
